FUNCTION_BLOCK TwoStateSwitch
VAR
	digitalInput : I_DigitalInput;
END_VAR

METHOD FB_init : BOOL
VAR_INPUT
	bInitRetains : BOOL; // if TRUE, the retain variables are initialized (warm start / cold start)
	bInCopyCode : BOOL;  // if TRUE, the instance afterwards gets moved into the copy code (online change)
	DigitalInput : I_DigitalInput;
END_VAR
this^.digitalInput := DigitalInput;
END_METHOD

PROPERTY PUBLIC IsOn : BOOL
GET
IsOn := digitalInput.State;
END_GET
END_PROPERTY

END_FUNCTION_BLOCK

(* stored: Version 1.1.0.1, ProductVersion 3.1.4024.5
   POU TwoStateSwitch: Id {ffe12da9-7ff2-45b0-85a9-aa27eb834c6f}, SpecialFunc None
   Method FB_init: Id {b4d5bf36-0426-48d4-b625-c2cbba624363}
   Property IsOn: Id {3bd96306-3c08-4246-91c1-4c4c1fbf93c8}
   Get Get: Id {d7869862-2daf-4ab1-9381-c5df95bd2c70} *)
